TYPE EL3002_HWTOPLC_PDOS :
	STRUCT
		
	
	Channel1 	AT %I* : EL3002_CHANNEL;
	Channel2 	AT %I* : EL3002_CHANNEL;



	END_STRUCT
END_TYPE

(* stored: Version 1.1.0.1
   DUT EL3002_HWTOPLC_PDOS: Id {bad867cf-9e39-4d3d-a83a-8c58e8b102b0} *)
